(* PLC project Sin nombre, Desconocido Sin nombre 1 *)
(* stored: creationDateTime 2022-09-29T00:46:02, modificationDateTime 2022-09-29T06:09:05 *)

PROGRAM Parcial1
  VAR
    Prendido AT %IX0.0 : BOOL;
  END_VAR
  VAR
    Reset : BOOL := FALSE;
  END_VAR
  VAR
    SensorCarroEntrada AT %IX0.1 : BOOL;
    SensorCarroSalida AT %IX0.2 : BOOL;
    RetirarTicket AT %IX0.3 : BOOL;
    ValidarTicket AT %IX0.4 : BOOL;
  END_VAR
  VAR
    IR_Reset : BOOL;
    Proceso1 : BOOL;
  END_VAR
  VAR
    Error1 AT %QX0.2 : BOOL;
    Error2 AT %QX0.3 : BOOL;
    PuertaEntrada AT %QX0.0 : BOOL;
    PuertaSalida AT %QX0.1 : BOOL;
  END_VAR
  VAR
    TON_Entrada : TIME;
    TON_Salida : TIME;
    ContadorEntrada : INT;
    ContadorSalida : INT;
    TON0 : TON;
    CTU0 : CTU;
    TON1 : TON;
    CTU1 : CTU;
  END_VAR
  VAR  (* added by the conversion: wires and edge detectors of the diagram *)
    R_TRIG1 : R_TRIG;
    R_TRIG2 : R_TRIG;
  END_VAR

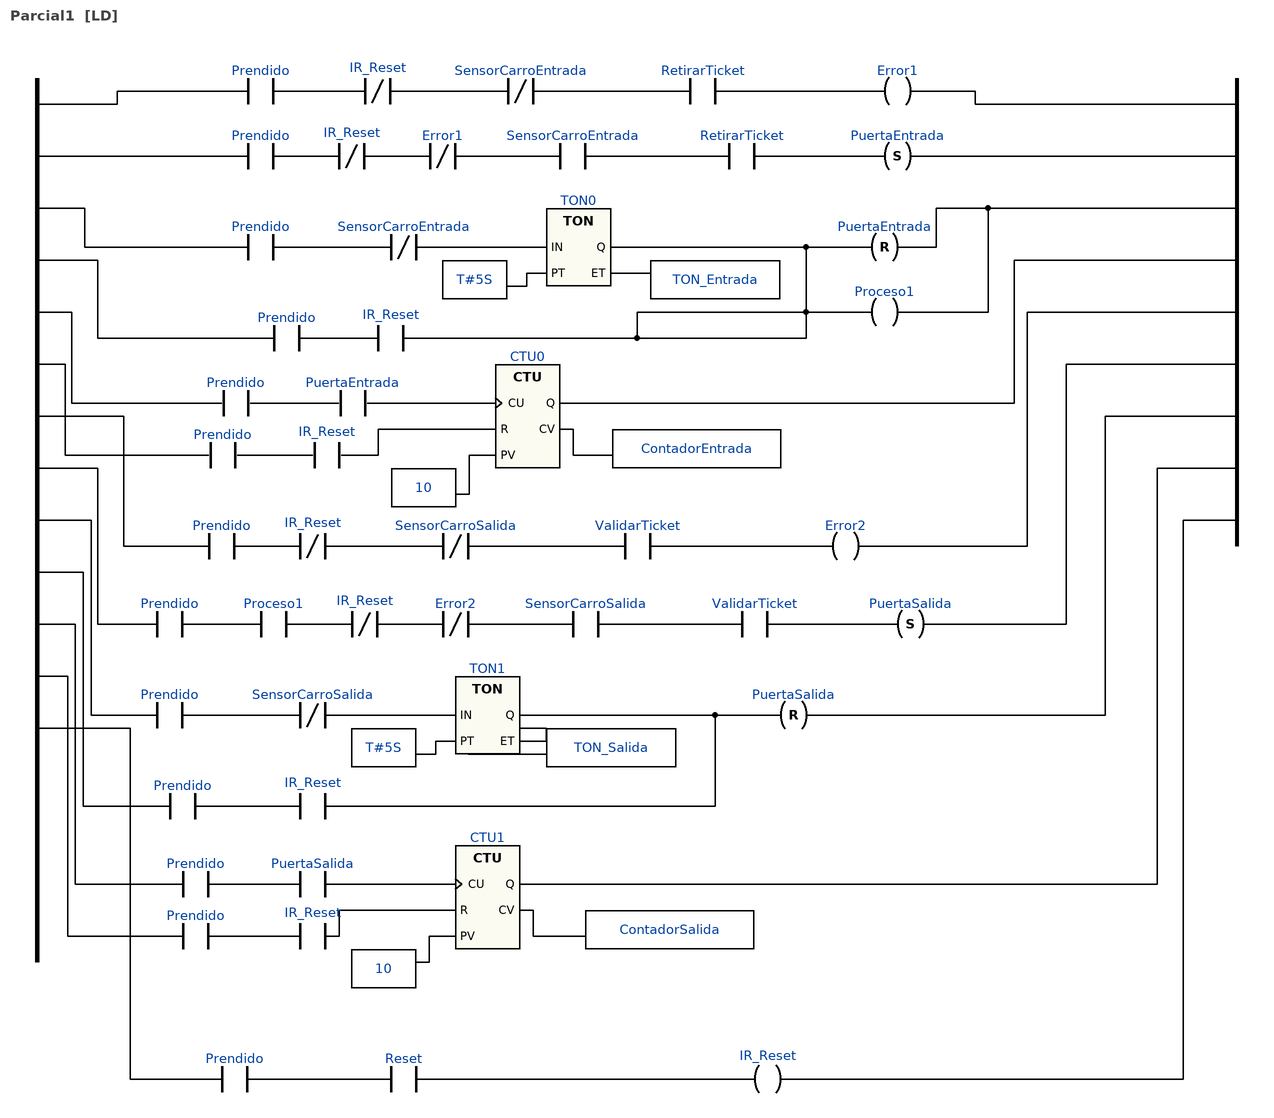
(* LD diagram, written out as Structured Text *)
Error1 := Prendido AND NOT IR_Reset AND NOT SensorCarroEntrada AND RetirarTicket;
IF Prendido AND NOT IR_Reset AND NOT Error1 AND SensorCarroEntrada AND RetirarTicket THEN PuertaEntrada := TRUE; END_IF;
TON0(IN := Prendido AND NOT SensorCarroEntrada, PT := T#5S);
IF TON0.Q OR Prendido AND IR_Reset THEN PuertaEntrada := FALSE; END_IF;
TON_Entrada := TON0.ET;
Proceso1 := Prendido AND IR_Reset OR TON0.Q;
R_TRIG1(CLK := Prendido AND PuertaEntrada);
CTU0(CU := R_TRIG1.Q, R := Prendido AND IR_Reset, PV := 10);
ContadorEntrada := CTU0.CV;
Error2 := Prendido AND NOT IR_Reset AND NOT SensorCarroSalida AND ValidarTicket;
IF Prendido AND Proceso1 AND NOT IR_Reset AND NOT Error2 AND SensorCarroSalida AND ValidarTicket THEN PuertaSalida := TRUE; END_IF;
TON1(IN := Prendido AND NOT SensorCarroSalida, PT := T#5S);
IF TON1.Q OR Prendido AND IR_Reset THEN PuertaSalida := FALSE; END_IF;
TON_Salida := TON1.ET;
R_TRIG2(CLK := Prendido AND PuertaSalida);
CTU1(CU := R_TRIG2.Q, R := Prendido AND IR_Reset, PV := 10);
ContadorSalida := CTU1.CV;
IR_Reset := Prendido AND Reset;
END_PROGRAM

CONFIGURATION Config0
  RESOURCE Res0 ON PLC
    TASK task0(INTERVAL := T#50ms, PRIORITY := 0);
    PROGRAM instance0 WITH task0 : Parcial1;
  END_RESOURCE
END_CONFIGURATION
